INTERFACE PUBLIC SuspendedCommands EXTENDS RunningStateCommands, HoldableStateCommands

METHOD PUBLIC Unsuspend
END_METHOD

END_INTERFACE

(* stored: Version 1.1.0.1, ProductVersion 3.1.4026.18
   Itf SuspendedCommands: Id {f31c0d5b-acac-0491-1bc4-9e5110404f07}
   Method Unsuspend: Id {199c3e50-b73d-0b1c-0fc2-c7e590019e1b} *)
